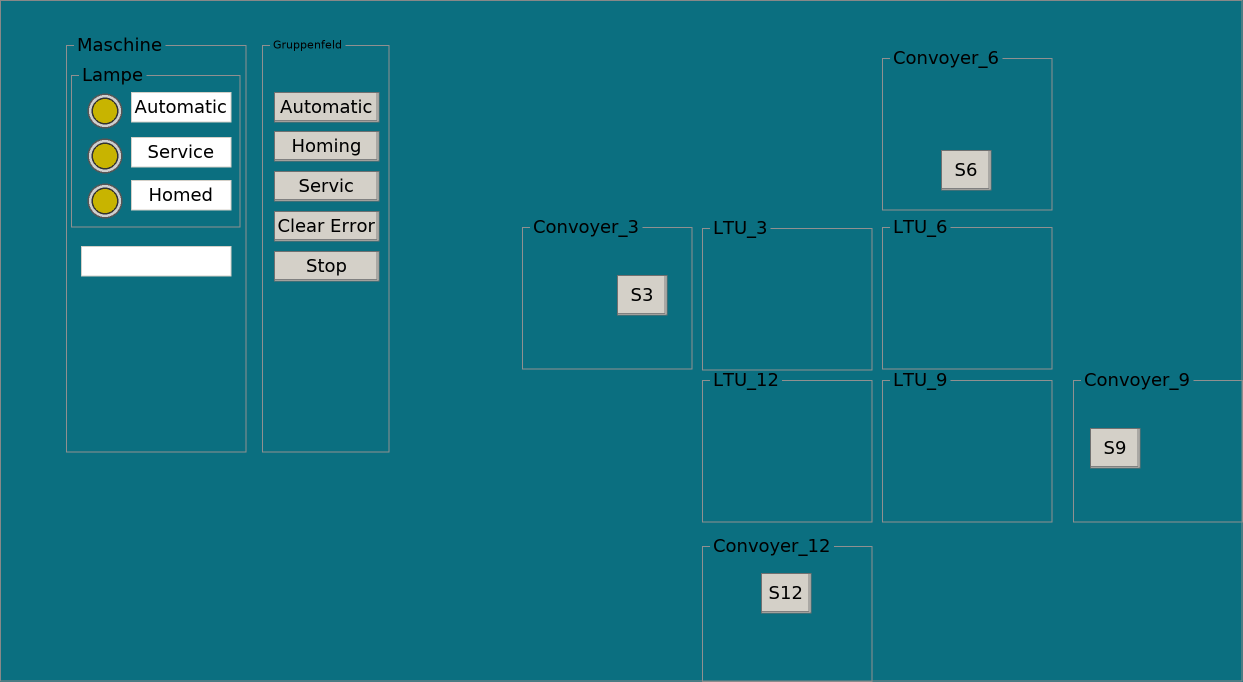
VISUALIZATION Visu_Customer  // 1243x682
    GroupBox (66,37 180x415), "Maschine"
        GroupBox (5,30 169x160), "Lampe"
            Lamp1 (14,114 40x40), style: Lamp-Lamp1-Yellow
            Lamp1 (14,69 40x40), style: Lamp-Lamp1-Yellow
            Lamp1 (14,24 40x40), style: Lamp-Lamp1-Yellow
            Textfield (60,25 100x30), "Automatic"
            Textfield (60,70 100x30), "Service"
            Textfield (60,113 100x30), "Homed"
        Textfield (15,209 150x30)
    GroupBox (262,37 127x415), "Gruppenfeld"
        Button (12,55 105x30), "Automatic"
        Button (12,94 105x30), "Homing"
        Button (12,134 105x30), "Servic"
        Button (12,174 105x30), "Clear Error"
        Button (12,214 105x30), "Stop"
    GroupBox (522,219 170x150), "Convoyer_3"
        Button (95,56 50x40), "S3"
    GroupBox (702,220 170x150), "LTU_3"
    GroupBox (882,219 170x150), "LTU_6"
    GroupBox (882,372 170x150), "LTU_9"
    GroupBox (702,372 170x150), "LTU_12"
    GroupBox (882,50 170x160), "Convoyer_6"
        Button (59,100 50x40), "S6"
    GroupBox (702,538 170x144), "Convoyer_12"
        Button (59,35 50x40), "S12"
    GroupBox (1073,372 170x150), "Convoyer_9"
        Button (17,56 50x40), "S9"
END_VISUALIZATION

(* stored: Version 1.1.0.1, ProductVersion 3.1.4026.18
   Visu Visu_Customer: Id {41bb52dc-3ba4-40b2-80e4-ac4579fbf1a3} *)
